(* IEC 61131-3 sources: com.logicals.lc3.webinar/usRTS_RPMControl_iSOC/src_FB_LIB_SAFE/Safe, 5 files *)

(* ---- TypeSAFEBOOL.iecst ---- *)
{ CustomImplementation }

NAMESPACE logicals.web.standard.safe

TYPE
	SAFEBOOL_Constant : BYTE(SAFEFALSE := 16#00, SAFETRUE := 16#AA);
	SAFEBOOL : BYTE := SAFEBOOL_Constant#SAFEFALSE;
END_TYPE

END_NAMESPACE

(* ---- TypeSAFEINT.iecst ---- *)
{ CustomImplementation }

NAMESPACE logicals.web.standard.safe

TYPE
	SAFEINT : INT := 0;
END_TYPE

END_NAMESPACE

(* ---- CheckSAFEBOOL.iecst ---- *)
NAMESPACE logicals.web.standard.safe

/* only a internal/private helper function - should not be public in a library */
FUNCTION CheckSAFEBOOL : BOOL
	VAR_INPUT
		IN : SAFEBOOL;
	END_VAR
	CheckSAFEBOOL := IN = SAFEBOOL_Constant#SAFEFALSE OR IN = SAFEBOOL_Constant#SAFETRUE;
END_FUNCTION

END_NAMESPACE

(* ---- IS.iecst ---- *)
NAMESPACE logicals.web.standard.safe

FUNCTION IS : BOOL
	VAR_INPUT
		In : SAFEBOOL;
	END_VAR
	IS := (In <> SAFEBOOL_Constant#SAFEFALSE);
END_FUNCTION

END_NAMESPACE

(* ---- IS_NOT.iecst ---- *)
NAMESPACE logicals.web.standard.safe

FUNCTION IS_NOT : BOOL
	VAR_INPUT
		In : SAFEBOOL;
	END_VAR
	IS_NOT := (In = SAFEBOOL_Constant#SAFEFALSE);
END_FUNCTION

END_NAMESPACE
